FUNCTION_BLOCK FB_SimpleFuse
VAR_INPUT
END_VAR
VAR_OUTPUT
END_VAR
VAR
	Chn1 : EL922x_ChannelBasic;
END_VAR

END_FUNCTION_BLOCK

(* stored: Version 1.1.0.1, ProductVersion 3.1.4024.5
   POU FB_SimpleFuse: Id {6ba8ae37-75f1-446b-9d7f-12fc08dcb036}, SpecialFunc None *)
